// TIA Portal V21 export
TYPE "OBJ_Washing_Step_V210_Type"
   STRUCT
      "w_Output Working 01" { S7_SetPoint := 'True'} : Word := W#16#0000;   // Output Working Data 1
      "w_Output Working 02" { S7_SetPoint := 'True'} : Word := W#16#0000;   // Output Working Data 2
      "w_Output Working 03" { S7_SetPoint := 'True'} : Word := W#16#0000;   // Output Working Data 3
      "w_Output Working 04" { S7_SetPoint := 'True'} : Word := W#16#0000;   // Output Working Data 4
      "i_Type Contition" { S7_SetPoint := 'True'} : Int;   // 0=Time 1=Wait Cond 2=Cnt 4=Speed 16=End Recipe
      "w_Waiting Condition" { S7_SetPoint := 'True'} : Word := W#16#0000;   // Waiting Condition
      w_SetPoint { S7_SetPoint := 'True'} : Int;   // Setpoint Data
      "w_Timer Jump" { S7_SetPoint := 'True'} : Int;   // Minimum Timer Adjustment
      "i_Step Description" { S7_SetPoint := 'True'} : Int;   // Text Number to Describe the Step
      "i_Step Image" { S7_SetPoint := 'True'} : Int;   // Image Number to Describe the Step
   END_STRUCT;
END_TYPE
